		This step we would save cycle time value (e.g. we not include saving data into cycle time )
		
*)
IF (Step(2150, TRUE, 'STOP MEASURE CT TRIGGER')) THEN
    //-------------------------------------    
    StopCleanCycleTime();
    StepCompleteWhen(TRUE);
    //-------------------------------------
END_IF

(*

	CLOSING DATA OPERATIONS
	Following methods provide process data manipulation for this controlled unit.
	Comment or uncomment according to your need.
*)
// Populates the information in the data header of this controlled unit (operations end time stamp, user info, etc)
// Typically used after all steps within the controlled unit are completed.
IF (_dataClose) THEN
    THIS^.DataEntityClose(5000, eDataEntityInvokeType.InvokeAndWaitDone, Station.ProcessDataManager.Data.CU00x.Header);
END_IF;

// Populates the information in the data header of this controlled unit (operations end time stamp, user info, etc)
// Typically used after all operation on the technology are completed.
// Input parameter eDataEntityInvokeType.InvokeOnly is used for speed up cycle(TRUE)
IF (_dataFinalize) THEN
    THIS^.DataEntityFinalize(5500, eDataEntityInvokeType.InvokeOnly, Station.ProcessDataManager.Data.CU00x.Header);
END_IF;

IF (Step(10000, TRUE, 'WAIT FOR PARALELL TASK TO FINISH')) THEN
    //-------------------------------------
    StepCompleteWhen(_paralellTask.Task.Done);

    IF _paralellTask.Task.Done THEN
        _paralellTask.Restore();
		
    END_IF
    //-------------------------------------	
END_IF

IF (Step(20000, _dataClose, 'WAIT FOR IF DATA FINALIZE IS DONE')) THEN
    //-------------------------------------
    StepCompleteWhen(Station.UpdateEntityTask.Done);
	CustomObserver.SetCycleId(Station.ProcessDataManager.Data._EntityId);
    //-------------------------------------	
END_IF



//monitor if conseccutive failures occur during automatic cycle. System monitor two basic types like are arbitrary failure in seqence, or  same(equal) failure in sequence
//if Number of allowed recurring failure is 0 , monitoring is inactive.
//Recurring failures are based on ErrorCodes in TcoComprehensiveResult.
//If error code in Same recurring failure is empty string ,monitorig of failure is not performed.
//Error code in Arbitrary Recuring failure is irelevant.    
THIS^.MonitorAnyRecurringFailure(22000,THIS^.Station._settings.AnyRecurringFailure>0 , Station.ProcessDataManager.Data.EntityHeader.Results);
THIS^.MonitorSameRecurringFailure(22100,THIS^.Station._settings.SameRecurringFailure>0 , Station.ProcessDataManager.Data.EntityHeader.Results);



IF (Step(30000, TRUE, 'LAST STEP')) THEN
    //-------------------------------------

		IF (_loop) THEN
			CompleteSequence();
		END_IF;


    //-------------------------------------	
END_IF

_paralellTask();
END_METHOD

METHOD PUBLIC OnStart
SUPER^.OnStart();
Station.GroundTask.Restore();
Station.ManualTask.Restore();
Station.GroundTask.CancelGround();
_paralellTask.Restore();
END_METHOD

(*~
	<docu>
		<summary>
			Loads process settings from the current process set into this controlled unit.
			The `StationProcessDataManager.Data` is populated by data from process settings.						
		</summary>
	</docu>
~*)
METHOD PairTag : BOOL
VAR_INPUT
	inStepID : INT;
END_VAR

VAR
	answer: TagsPairing;
	_addNewTag: BOOL;
	dialogAnswer: eDialogAnswer;
END_VAR
IF (Step(inStepID, _tagsPairing, '<#PAIR TAG WITH ASSIGNED VALUE EXAMPLE#>')) THEN
    //-------------------------------------
	_addNewTag:=FALSE;

	answer:= Station.Components.PairTagTask.Answer;
	//this field may be assigned by unique ID of rfid chip , or dmc code.The PairTagTask provide answer where is assigned user defined value for this unique ID value.
	//If not, there may be diferent scenarios defined. See example bellow.
	_reqKey:='123456789';				   
	 IF Station.Components.PairTagTask.Run(inMode:=eTagPairingMode.GetTag, inKey:=_reqKey ,inAssignedValue:='').Invoke().Done	 THEN
		
		IF  answer.Answer =eTagPairingAnswer.TagFound 
			 THEN
			Station.ProcessDataManager.Data.EntityHeader.Carrier := answer.AssignedValue;
			CompleteStep();
			Station.Components.PairTagTask.Restore();
		
		ELSIF  answer.Answer = eTagPairingAnswer.TagFoundInactive THEN
			IF (_dialog.Show()
			   .WithCaption('<#Pairing Tag#>')
			   .WithText(_sb.Clear().Append('<#Founded tag#> ').Append(_reqKey).Append(' <#is inactive!#> ').Append(Station.Components.PairTagTask.AnswerInstruction).ToString() )
				.WithOk().Answer = TcoCore.eDialogAnswer.OK) THEN;
				;// Founded tag is Inactive. Probably carier(pallete) was disasbled due produced many errors.Se  here you can write diferent scenario ( leave it with current state , provide ground etc)	 
		
				//Station.GroundTask.Task.Invoke();
			   
			End_if;
		
		ELSIF  answer.Answer = eTagPairingAnswer.TagFoundAssignedValueEmpty THEN
			  IF (_dialog.Show()
			   .WithCaption('<#Pairing Tag#>')
			   .WithText(_sb.Clear().Append('<#Tag#> ').Append(_reqKey).Append(' <#is founded but assigned value is empty! Would you like continue?#> ').Append(Station.Components.PairTagTask.AnswerInstruction).ToString() )
				.WithYesNo().Answer = TcoCore.eDialogAnswer.Yes) THEN;
				CompleteStep();
				Station.Components.PairTagTask.Restore();
			END_IF;
		   
		ELSIF  answer.Answer = eTagPairingAnswer.TagNotFound THEN
			  IF (_dialog.Show()
			   .WithCaption('<#Pairing Tag#>')
			   .WithText(_sb.Clear().Append('<#Tag#> ').Append(_reqKey).Append(' <#is not founded ! Would you like assign right now?#> ').Append(Station.Components.PairTagTask.AnswerInstruction).ToString() )
				.WithYesNo().Answer = TcoCore.eDialogAnswer.Yes) THEN;
				_addNewTag:=TRUE;
				CompleteStep();
				Station.Components.PairTagTask.Restore();
			END_IF;
	
		
			ELSIF  answer.Answer = eTagPairingAnswer.EmptyCollection THEN
			  IF (_dialog.Show()
			   .WithCaption('<#Pairing Tag#>')
			   .WithText(_sb.Clear().Append('<#Tag#> ').Append(_reqKey).Append(' <#is not founded due collection is empty ! Would you like assign right now?#> ').Append(Station.Components.PairTagTask.AnswerInstruction).ToString() )
				.WithYesNo().Answer = TcoCore.eDialogAnswer.Yes) THEN;
				_addNewTag:=TRUE;
				CompleteStep();
				Station.Components.PairTagTask.Restore();
			END_IF;
		End_if;
			
	END_IF		    				
    //-------------------------------------
END_IF

IF (Step(inStepID+10, _tagsPairing AND _addNewTag, '<#ADD NEW TAG  EXAMPLE#>')) THEN
    //-------------------------------------
	
	answer:= Station.Components.PairTagTask.Answer;
	//this field may be assigned by unique ID of rfid chip , or dmc code.The PairTagTask provide answer where is assigned user defined value for this unique ID value.
	//If not, there may be diferent scenarios defined. See example bellow.
	_reqKey:='123456789';		
	_reqAssignedValue := 'CustomIdExample123';	   
	 IF Station.Components.PairTagTask.Run(inMode:=eTagPairingMode.AddTag, inKey:=_reqKey, inAssignedValue:=_reqAssignedValue).Invoke().Done	 THEN
		
		IF  answer.Answer =eTagPairingAnswer.TagAddedSuccessfully 
			 THEN
			Station.ProcessDataManager.Data.EntityHeader.Carrier := answer.AssignedValue;
			CompleteStep();
			Station.Components.PairTagTask.Restore();
		END_IF;
	ELSIF  answer.Answer = eTagPairingAnswer.TagAlreadyExist THEN
		IF (_dialog.Show()
	       .WithCaption('<#Adding Tag#>')
		   .WithText(_sb.Clear().Append('<#Tag#> ').Append(_reqKey).Append(' <#already exist!#> ').Append(Station.Components.PairTagTask.AnswerInstruction).ToString() )
			.WithOk().Answer = TcoCore.eDialogAnswer.OK) THEN;
			;// Founded tag is Inactive. Probably carier(pallete) was disasbled due produced many errors.Se  here you can write diferent scenario ( leave it with current state , provide ground etc)	 
	
		 	//Station.GroundTask.Task.Invoke();
		   
		End_if;
	
	ELSIF  answer.Answer = eTagPairingAnswer.TagAddedNotSuccessfuly THEN
			dialogAnswer := _dialog.Show()
	       .WithCaption('<#Pairing Tag#>')
		   .WithText(_sb.Clear().Append('<#Tag#> ').Append(_reqKey).Append(' <#was not founnd! Would you like still like to continue?#> ').Append(Station.Components.PairTagTask.AnswerInstruction).ToString() )
			.WithYesNo().Answer;
			
	      IF (dialogAnswer= TcoCore.eDialogAnswer.Yes) THEN;
			CompleteStep();
			Station.Components.PairTagTask.Restore();
		END_IF;
		   

			
	END_IF		    				
    //-------------------------------------
END_IF
END_METHOD

METHOD SingleExample : BOOL
VAR_INPUT
		inStepID : INT;
END_VAR

IF (Step(inStepID, TRUE, 'SINGLE INSPECTION')) THEN
    //-------------------------------------    
	Station.ProcessDataManager.Data.CU00x.BoltPresenceInspector.Data.FailureDescription:='BoltPresenceInspector error';
    Station.ProcessDataManager.Data.CU00x.BoltPresenceInspector.WithCoordinator(THIS^)
        .Inspect(_inspectionResult)
        .UpdateComprehensiveResult(Station.ProcessDataManager.Data.EntityHeader.Results)
        .OnFail().Dialog(inStepID+10);
    //-------------------------------------
END_IF

// with checking if specific inspector is overinspected
IF (Step(inStepID+10, TRUE, 'SINGLE ANALOGUE INSPECTION')) THEN
//-------------------------------------
	Station.ProcessDataManager.Data.CU00x.BoltDimensionPresenceInspector.Data.FailureDescription:='BoltDimensionPresenceInspector error';
	Station.ProcessDataManager.Data.CU00x.BoltDimensionPresenceInspector.Data.NumberOfAllowedRetries:=100;
	IF NOT Station.ProcessDataManager.Data.CU00x.BoltDimensionPresenceInspector.OverInspected THEN
	
		Station.ProcessDataManager.Data.CU00x.BoltDimensionPresenceInspector.WithCoordinator(THIS^)
			.Inspect(_inspectionDimensionResult)
			.WithDescription()
			.UpdateComprehensiveResult(Station.ProcessDataManager.Data.EntityHeader.Results)
			.OnFail().Retry(inStepID+20);
	ELSE
	 	RequestStep(RESTORE_STEP_ID);	
	END_IF
//-------------------------------------
END_IF;

IF (Step(inStepID+20, TRUE, 'DONE')) THEN
//-------------------------------------
		CompleteStep();
//-------------------------------------
END_IF;
END_METHOD

PROPERTY Station : REFERENCE TO CU00x
GET
VAR
    _station : POINTER TO CU00x;
END_VAR
IF __QUERYPOINTER(Parent, _station) THEN // Check if _Parent is Station001
    Station REF= _station^;              // If the check is successful dereference a pointer. simlar to THIS^ or SUPER^
END_IF
END_GET
END_PROPERTY

END_FUNCTION_BLOCK

// ---- Technology/CU00x/Safety/Suspend/CU00xSuspendTask.TcPOU
FUNCTION_BLOCK CU00xSuspendTask EXTENDS CUBaseSuspend IMPLEMENTS ICUTask
VAR

END_VAR

Run();

(*~
	<docu>
		<summary>
			Main method of the sequener. Custom code needs to be placed here. The sequencer is executed by call of **Instance.Run()** method.
			This method is abstract, and it must be overridden in derived block.
		</summary>
	</docu>
~*)
METHOD PROTECTED Main : BOOL
(*

	SUSPEND PROCESS 
	Following steps provide suspend actions for this controlled unit.
	Add components add write customized sequence according to your need.
*)

		
//
IF (Step(100, TRUE, '<#WAITING FOR START#>')) THEN
    //-------------------------------------    

    StepCompleteWhen(TRUE);
    //-------------------------------------
END_IF

//HERE  YOU CAN WRITE  WHAT IS NECESSARY 
//TO SUPSEND  PROCESS..... TO INTERUPT SAFETY

IF (Step(1000, TRUE, '<#SUSPENDING COMPONENTS#>')) THEN
 	//-------------------------------------    
	//StepCompleteWhen(Station.AutomatTask.CurrentStep.Status <> eStepStatus.Running);
		
    StepCompleteWhen( CurrentStep.Duration >= T#3000MS);
    //-------------------------------------
END_IF

IF (Step(30000, TRUE, 'SUSPEND DONE')) THEN
    //-------------------------------------
		
        THIS^._done:=TRUE;
		THIS^.Task.DoneWhen(TRUE);
	
   
    //-------------------------------------	
END_IF
END_METHOD

METHOD PUBLIC OnStart
SUPER^.OnStart();
Station.RecoverTask.Restore();
END_METHOD

PROPERTY Station : REFERENCE TO CU00x
GET
VAR
    _station : POINTER TO CU00x;
END_VAR
IF __QUERYPOINTER(Parent, _station) THEN // Check if _Parent is Station001
    Station REF= _station^;              // If the check is successful dereference a pointer. simlar to THIS^ or SUPER^
END_IF
END_GET
END_PROPERTY

END_FUNCTION_BLOCK

// ---- Technology/CU00x/Safety/Recover/CU00xRecoverTask.TcPOU
FUNCTION_BLOCK CU00xRecoverTask EXTENDS CUBaseRecover IMPLEMENTS ICUTask
VAR

END_VAR

Run();

(*~
	<docu>
		<summary>
			Main method of the sequener. Custom code needs to be placed here. The sequencer is executed by call of **Instance.Run()** method.
			This method is abstract, and it must be overridden in derived block.
		</summary>
	</docu>
~*)
METHOD PROTECTED Main : BOOL
(*

	RECOVER PROCESS 
	Following steps provide recover action for this controlled unit.
	Add components add write customized sequence according to your need.
*)

		
//
IF (Step(100, TRUE, '<#WAITING FOR START#>')) THEN
    //-------------------------------------    

    StepCompleteWhen(TRUE);
    //-------------------------------------
END_IF

//HERE  YOU CAN WRITE  WHAT IS NECESSARY 
//TO RECOVER AFTER INTERUPTED PROCESS.....

IF (Step(1000, TRUE, '<#RECOVER ANY COMPONENTS#>')) THEN
    //-------------------------------------    

    StepCompleteWhen(CurrentStep.Duration >= T#3000MS);
    //-------------------------------------
END_IF

IF (Step(30000, TRUE, 'RECOVER DONE')) THEN
    //-------------------------------------
		
        this^._done:=true;
		THIS^.Task.DoneWhen(TRUE);
		
   
    //-------------------------------------	
END_IF
END_METHOD

METHOD PUBLIC OnStart
SUPER^.OnStart();
Station.SuspendTask.Restore();
END_METHOD

PROPERTY Station : REFERENCE TO CU00x
GET
VAR
    _station : POINTER TO CU00x;
END_VAR
IF __QUERYPOINTER(Parent, _station) THEN // Check if _Parent is Station001
    Station REF= _station^;              // If the check is successful dereference a pointer. simlar to THIS^ or SUPER^
END_IF
END_GET
END_PROPERTY

END_FUNCTION_BLOCK
